FUNCTION_BLOCK Lincon
VAR_INPUT
	Enable:BOOL; (**)
	Input:INT; (**)
	Multiplier:INT; (**)
	DIvisor:INT; (**)
	Offset:INT; (**)
END_VAR
VAR_OUTPUT
	Out:INT; (**)
END_VAR
VAR
END_VAR
VAR
	Mul_r:REAL;
	Div_r:REAL;
	In_r:REAL;
	Out_r:REAL;
	Err_b:BOOL;
END_VAR
VAR // added by the converter: edge detectors and wires of the graphical bodies
    _w1, _w2, _w4, _w8, _w10 : REAL;
    _w3, _w5, _w6, _w7, _w12, _w16, _w18, _w19, _w20, _w22 : BOOL;
    _w9, _w21 : DINT;
    _w11, _w13, _w14, _w15 : INT;
    _w17, _w23 : ANY;
END_VAR

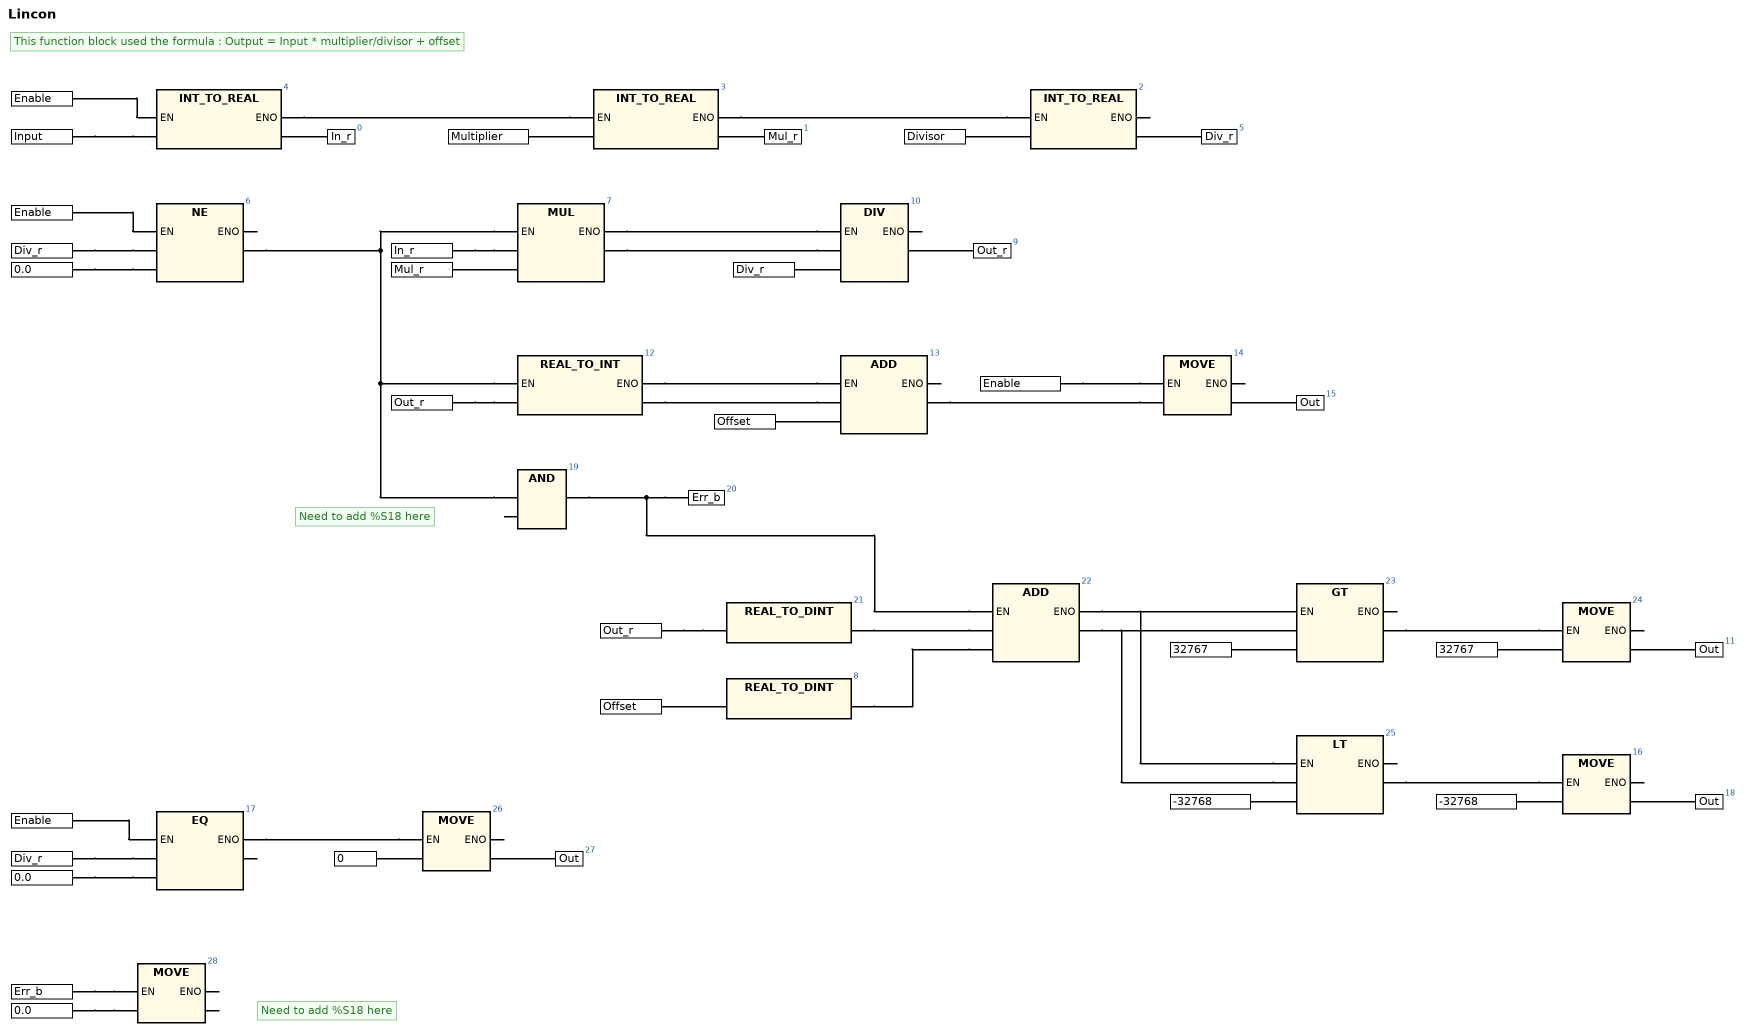
In_r := _w1;
Mul_r := _w2;
IF _w3 THEN _w4 := INT_TO_REAL(Divisor); END_IF
_w3 := _w5;
IF _w3 THEN _w2 := INT_TO_REAL(Multiplier); END_IF
// This function block used the formula : Output = Input * multiplier/divisor + offset
_w5 := Enable;
IF _w5 THEN _w1 := INT_TO_REAL(Input); END_IF
Div_r := _w4;
IF Enable THEN _w6 := Div_r <> 0.0; END_IF
_w7 := _w6;
IF _w7 THEN _w8 := In_r * Mul_r; END_IF
_w9 := REAL_TO_DINT(Offset);
Out_r := _w10;
IF _w7 THEN _w10 := _w8 / Div_r; END_IF
Out := _w11;
_w12 := _w6;
IF _w12 THEN _w13 := REAL_TO_INT(Out_r); END_IF
IF _w12 THEN _w14 := _w13 + Offset; END_IF
IF Enable THEN _w15 := _w14; END_IF
Out := _w15;
IF _w16 THEN _w17 := -32768; END_IF
_w18 := Enable;
IF _w18 THEN (* Div_r = 0.0; result not used *) END_IF
Out := _w17;
_w19 := _w6 AND ???;
// Need to add %S18 here
Err_b := _w19;
_w20 := _w19;
IF _w20 THEN _w21 := REAL_TO_DINT(Out_r) + _w9; END_IF
IF _w20 THEN _w22 := _w21 > 32767; END_IF
IF _w22 THEN _w11 := 32767; END_IF
IF _w20 THEN _w16 := _w21 < -32768; END_IF
IF _w18 THEN _w23 := 0; END_IF
Out := _w23;
// Need to add %S18 here
IF Err_b THEN (* 0.0; result not used *) END_IF

END_FUNCTION_BLOCK

(* stored: Version 1.1.0.1, ProductVersion 3.1.4024.0
   POU Lincon: Id {5dfe4370-8e73-4ee7-bda7-e92777189b08}, SpecialFunc None *)
